{attribute 'qualified_only'}
VAR_GLOBAL
END_VAR

(* stored: Version 1.1.0.1, ProductVersion 3.1.4024.16
   GVL GVL: Id {8da3d8d1-59ea-492c-bb1b-f77e34f6aa4a} *)
